FUNCTION_BLOCK ROBOTFB (* JADE WORKER *)
  (* Standard: 61499-1 *)
  (* Version 1.0, 2014-04-22, Ahmed, Fraunhofer IGD *)
  (* Compiler header: package fb.rt; *)
  (* Compiler Java Sun JDK 1.5.0 *)
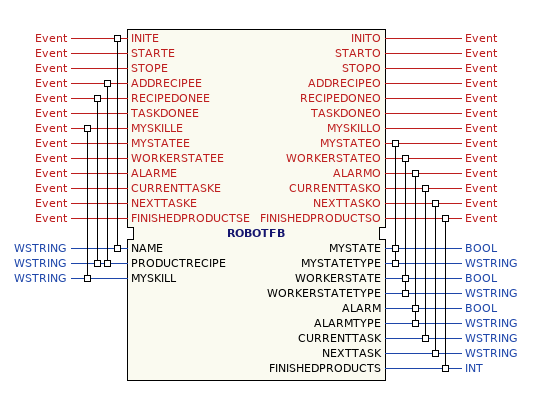
  EVENT_INPUT
    INITE WITH NAME;
    STARTE; (* Normal Execution Request *)
    STOPE;
    ADDRECIPEE WITH PRODUCTRECIPE;
    RECIPEDONEE WITH PRODUCTRECIPE;
    TASKDONEE;
    MYSKILLE WITH MYSKILL;
    MYSTATEE;
    WORKERSTATEE;
    ALARME;
    CURRENTTASKE;
    NEXTTASKE;
    FINISHEDPRODUCTSE;
  END_EVENT
  EVENT_OUTPUT
    INITO;
    STARTO; (* Execution Confirmation *)
    STOPO;
    ADDRECIPEO;
    RECIPEDONEO;
    TASKDONEO;
    MYSKILLO;
    MYSTATEO WITH MYSTATE, MYSTATETYPE;
    WORKERSTATEO WITH WORKERSTATE, WORKERSTATETYPE;
    ALARMO WITH ALARM, ALARMTYPE;
    CURRENTTASKO WITH CURRENTTASK;
    NEXTTASKO WITH NEXTTASK;
    FINISHEDPRODUCTSO WITH FINISHEDPRODUCTS;
  END_EVENT
  VAR_INPUT
    NAME : WSTRING;
    PRODUCTRECIPE : WSTRING;
    MYSKILL : WSTRING;
  END_VAR
  VAR_OUTPUT
    MYSTATE : BOOL;
    MYSTATETYPE : WSTRING;
    WORKERSTATE : BOOL;
    WORKERSTATETYPE : WSTRING;
    ALARM : BOOL;
    ALARMTYPE : WSTRING;
    CURRENTTASK : WSTRING;
    NEXTTASK : WSTRING;
    FINISHEDPRODUCTS : INT;
  END_VAR
END_FUNCTION_BLOCK
